FUNCTION_BLOCK FB_PISTON
VAR_INPUT
	eSTATE:E_STATE:=E_STATE.uninit;
	sSTATE:STRING:='UNINIT';
	sNAME:STRING;
	bLOCAL_MANUAL: BOOL:=FALSE;
	pist_TYPE: E_PISTON_TYPE;
	pist_STATE: E_PISTON_STATE:=E_PISTON_STATE.uninit;
	rOPEN_TIME: TIME;
	rCLOSE_TIME: TIME;
	rOPEN_TIMEOUT: TIME;
	tCLOSE_TIMEOUT: TIME;
	bOPEN_LIMIT: BOOL;
	bCLOSED_LIMIT: BOOL;
	bOPEN_CMD: BOOL;
	bCLOSE_CMD: BOOL;
	bOPEN_SWR: BOOL;
	bCLOSE_SWR: BOOL;
	bCONDITION: BOOL:=TRUE;
	bLOCAL_RESET:BOOL;
END_VAR
VAR_OUTPUT
	bOPEN_VALVE: BOOL;
	bCLOSE_VALVE: BOOL;
	bBUSY:BOOL;
	bOPENED:BOOL;
	bCLOSED:BOOL;
	bERROR:BOOL:=FALSE;
END_VAR
VAR
	T_OPEN: TON;
	T_OPEN_TIMEOUT: TON;
	T_CLOSE: TON;
	T_CLOSE_TIMEOUT: TON;
	bOPEN_DEFAULT: BOOL:=FALSE;
	bFIRST_DONE: BOOL:=FALSE;
	
END_VAR

T_OPEN(IN:= bOPEN_CMD, PT:=rOPEN_TIME , Q=> , ET=> );
T_CLOSE(IN:=  NOT bOPEN_CMD, PT:=rCLOSE_TIME , Q=> , ET=> );
T_OPEN_TIMEOUT(IN:= bOPEN_CMD , PT:= rOPEN_TIMEOUT, Q=> , ET=> );
T_CLOSE_TIMEOUT(IN:=  NOT bOPEN_CMD , PT:= tCLOSE_TIMEOUT, Q=> , ET=> );

IF bLOCAL_RESET THEN//========================== RESET================
	bLOCAL_RESET:=FALSE;
	pist_STATE:=E_PISTON_STATE.uninit;
END_IF

IF NOT bLOCAL_MANUAL THEN//====================== MANUAL ==============
	bOPEN_CMD:=bOPEN_SWR;
END_IF

IF NOT bFIRST_DONE THEN  // ============== check default mode ===============
	bFIRST_DONE:=TRUE;
	IF bOPEN_DEFAULT THEN
		bOPEN_CMD:=TRUE;
	ELSE
		bOPEN_CMD:=FALSE;
	END_IF
END_IF
//================================================== UNINIT =====================================================
CASE pist_STATE OF
	E_PISTON_STATE.uninit:
		eSTATE:=E_STATE.uninit;
		bERROR:=FALSE;
		IF bOPEN_CMD  THEN
			bOPEN_VALVE:=TRUE;
			bCLOSE_VALVE:=FALSE;
			pist_STATE:=E_PISTON_STATE.opening;
		ELSE
			bOPEN_VALVE:=FALSE;
			bCLOSE_VALVE:=TRUE;
			pist_STATE:=E_PISTON_STATE.closing;
		END_IF
//================================================== OPENING =====================================================
	E_PISTON_STATE.opening:
	eSTATE:=E_STATE.busy;
	sSTATE:='OPENING';
	bBUSY:=TRUE; bOPENED:=FALSE; bCLOSED:=FALSE;
	CASE pist_TYPE OF//------------------------------no sensors
		E_PISTON_TYPE.NO_SENSORS:
		IF T_OPEN.Q THEN
			pist_STATE:=E_PISTON_STATE.opened;
		END_IF
		//----------------------------- both sensors
		E_PISTON_TYPE.BOTH:
		IF bOPEN_LIMIT THEN
			pist_STATE:=E_PISTON_STATE.opened;
		END_IF
		IF T_OPEN_TIMEOUT.Q THEN
			bOPEN_CMD:=FALSE;
			aPISTON_ERROR();
			pist_STATE:=E_PISTON_STATE.error;
		END_IF
		//----------------------------- only open sensor
		E_PISTON_TYPE.ONLY_OPEN:
		IF bOPEN_LIMIT THEN
			pist_STATE:=E_PISTON_STATE.opened;
		END_IF
		IF T_OPEN_TIMEOUT.Q THEN
			bOPEN_CMD:=FALSE;
			aPISTON_ERROR();
			pist_STATE:=E_PISTON_STATE.error;
		END_IF
		//----------------------------- only close sensor
		E_PISTON_TYPE.ONLY_CLOSE:
		IF T_OPEN.Q THEN
			pist_STATE:=E_PISTON_STATE.opened;
		END_IF
	END_CASE
//================================================== CLOSING =====================================================	
	E_PISTON_STATE.closing:
	eSTATE:=E_STATE.busy;
	sSTATE:='CLOSING'; bOPENED:=FALSE; bCLOSED:=FALSE;
	bBUSY:=TRUE;
	CASE pist_TYPE OF//--------------------------------------- no sensors
		E_PISTON_TYPE.NO_SENSORS:
		IF T_CLOSE.Q THEN
			pist_STATE:=E_PISTON_STATE.closed;
		END_IF
		//-------------------------------------- both sensors
		E_PISTON_TYPE.BOTH:
		IF bCLOSED_LIMIT THEN
			pist_STATE:=E_PISTON_STATE.closed;
		END_IF
		IF T_CLOSE_TIMEOUT.Q THEN
			bOPEN_CMD:=TRUE;
			pist_STATE:=E_PISTON_STATE.error;
		END_IF
		//-------------------------------------- only close sensor
		E_PISTON_TYPE.ONLY_CLOSE:
		IF bCLOSED_LIMIT THEN
			pist_STATE:=E_PISTON_STATE.closed;
		END_IF
		IF T_CLOSE_TIMEOUT.Q THEN
			bOPEN_CMD:=TRUE;
			aPISTON_ERROR();
			pist_STATE:=E_PISTON_STATE.error;
		END_IF
		//----------------------------- only close sensor
		E_PISTON_TYPE.ONLY_OPEN:
		IF T_CLOSE.Q THEN
			pist_STATE:=E_PISTON_STATE.closed;
		END_IF
	END_CASE
//================================================== OPENED =====================================================	
	E_PISTON_STATE.opened:
	eSTATE:=E_STATE.ready;
	sSTATE:='OPENED';
	bBUSY:=FALSE; bOPENED:=TRUE; bCLOSED:=FALSE;
	IF NOT bOPEN_CMD  THEN
		pist_STATE:=E_PISTON_STATE.closing;
		bOPEN_VALVE:=FALSE;
		bCLOSE_VALVE:=TRUE;
	END_IF
	CASE pist_TYPE OF
		//-------------------------------------- both sensors
		E_PISTON_TYPE.BOTH:
		IF NOT bOPEN_LIMIT THEN
			bOPEN_CMD:=FALSE;
			aPISTON_ERROR();
			pist_STATE:=E_PISTON_STATE.error;
		END_IF
		//-------------------------------------- only open sensor
		E_PISTON_TYPE.ONLY_OPEN:
		IF NOT bOPEN_LIMIT THEN
			bOPEN_CMD:=FALSE;
			aPISTON_ERROR();
			pist_STATE:=E_PISTON_STATE.error;
		END_IF
	END_CASE
//================================================== CLOSED =====================================================	
	E_PISTON_STATE.closed:
	eSTATE:=E_STATE.ready;
	sSTATE:='CLOSED';
	bBUSY:=FALSE; bOPENED:=FALSE; bCLOSED:=TRUE;
	IF bOPEN_CMD  THEN
		pist_STATE:=E_PISTON_STATE.opening;
		bOPEN_VALVE:=TRUE;
		bCLOSE_VALVE:=FALSE;
	END_IF
	CASE pist_TYPE OF
		//-------------------------------------- both sensors
		E_PISTON_TYPE.BOTH:
		IF NOT bCLOSED_LIMIT THEN
			bOPEN_CMD:=TRUE;
			aPISTON_ERROR();
			pist_STATE:=E_PISTON_STATE.error;
		END_IF
		//-------------------------------------- only close sensor
		E_PISTON_TYPE.ONLY_CLOSE:
		IF NOT bCLOSED_LIMIT THEN
			bOPEN_CMD:=TRUE;
			aPISTON_ERROR();
			pist_STATE:=E_PISTON_STATE.error;
		END_IF
	END_CASE
//================================================== ERROR =====================================================	
	E_PISTON_STATE.error:
	eSTATE:=E_STATE.error;
	sSTATE:='ERROR';
	bERROR:=TRUE;
	//
END_CASE

ACTION aCLOSE:
bOPEN_SWR:=FALSE;
END_ACTION

ACTION aHOME:
IF bOPEN_DEFAULT THEN
	bOPEN_SWR:=TRUE;
ELSE
	bOPEN_SWR:=FALSE;
END_IF
END_ACTION

ACTION aOPEN:
bOPEN_SWR:=TRUE;
END_ACTION

ACTION aPISTON_ERROR:
gEventType:= 'piston Alarm'; 
gEventSeverity:= 'Error';

gEventName:= sNAME;
IF pist_STATE=E_PISTON_STATE.opening  THEN
	gEventText:='piston opening';
	gEventIdentity:=1001;
END_IF
IF pist_STATE=E_PISTON_STATE.closing THEN
	gEventText:='piston closing';
	gEventIdentity:=1002;
END_IF
IF pist_STATE=E_PISTON_STATE.closed THEN
	gEventText:='piston closed';
	gEventIdentity:=1003;
END_IF
IF pist_STATE=E_PISTON_STATE.opened THEN
	gEventText:='piston opened';
	gEventIdentity:=1004;
END_IF
fbEventLogger.mAdd();
END_ACTION

ACTION aRESET:
bLOCAL_RESET:=TRUE;
END_ACTION

END_FUNCTION_BLOCK

(* stored: Version 1.1.0.1, ProductVersion 3.1.4024.12
   POU FB_PISTON: Id {f4523f62-f900-4afa-86ce-0e9446376750}, SpecialFunc None
   Action aCLOSE: Id {b1f4e35c-084e-407f-83a6-be1401f028cb}
   Action aHOME: Id {61cd54f0-31ef-41dc-b8af-f4a12fbdd7c4}
   Action aOPEN: Id {9c0def1d-a187-4f8f-b5bd-4536b7394c6f}
   Action aPISTON_ERROR: Id {1b759e5b-d5dc-4ee8-b4b9-3114018bbeff}
   Action aRESET: Id {04605110-f2be-4812-bdc3-32e8c11c9c1a} *)
